Yaskawa INFORM job: LONGPIPE_1.JBI

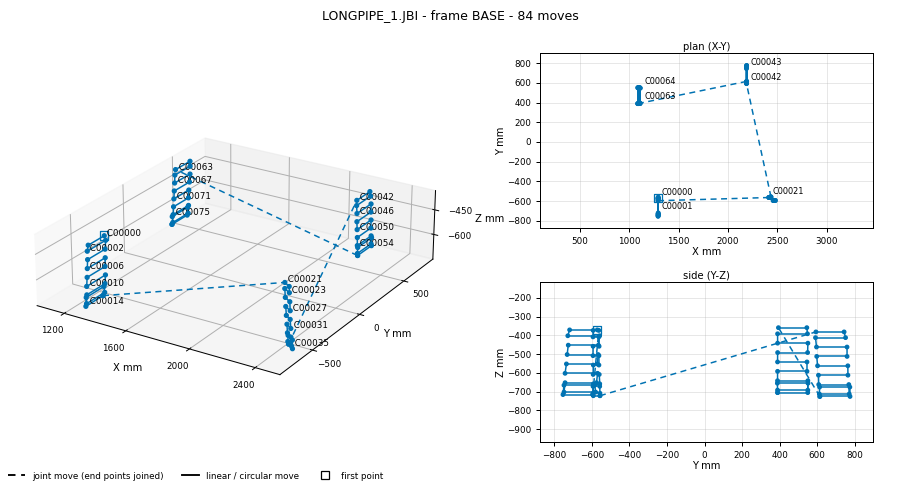
[picture p0: tool path of LONGPIPE_1.JBI in frame BASE, 84 of 89 moves have a stored position in this frame; points joined in program order, loops and branches not executed]
/JOB
//NAME LONGPIPE_1
//POS
///NPOS 84,0,84,0,0,0
///TOOL 1
///POSTYPE BASE
///RECTAN
///RCONF 1,0,0,0,0,0,0,0,0,0,0,0,0,0,0,0,0,0,0,0,0,0,0,0
C00000=1293.713569,-571.374698,-371.239941,175.000000,-89.999999,5.000000
C00001=1293.713569,-718.549324,-371.239941,175.000000,-89.999999,5.000000
C00002=1293.518411,-728.243914,-402.544866,175.000000,-89.999999,5.000000
C00003=1293.518411,-558.764125,-402.544866,175.000000,-89.999999,5.000000
C00004=1292.393979,-565.555949,-452.544866,175.000000,-89.999999,5.000000
C00005=1292.393979,-725.875043,-452.544866,175.000000,-89.999999,5.000000
C00006=1292.721121,-731.714794,-502.544866,175.000000,-89.999999,5.000000
C00007=1292.721121,-566.567624,-502.544866,175.000000,-89.999999,5.000000
C00008=1292.721835,-570.937787,-552.544866,175.000000,-89.999999,5.000000
C00009=1292.721835,-735.641722,-552.544866,175.000000,-89.999999,5.000000
C00010=1293.523260,-742.896244,-602.544866,175.000000,-89.999999,5.000000
C00011=1293.523260,-569.798478,-602.544866,175.000000,-89.999999,5.000000
C00012=1292.629099,-575.385878,-652.544866,175.000000,-89.999999,5.000000
C00013=1292.629099,-742.820182,-652.544866,175.000000,-89.999999,5.000000
C00014=1292.888223,-748.485672,-702.544866,175.000000,-89.999999,5.000000
C00015=1292.888223,-580.024935,-702.544866,175.000000,-89.999999,5.000000
C00016=1292.167541,-584.742252,-665.942326,180.000000,-60.000000,0.000000
C00017=1292.167541,-748.713534,-665.942326,180.000000,-60.000000,0.000000
C00018=1292.184485,-754.080694,-715.942326,180.000000,-60.000000,0.000000
C00019=1292.184485,-595.509845,-715.942326,180.000000,-60.000000,0.000000
C00020=1292.184485,-595.509845,-715.942326,180.000000,-60.000000,0.000000
C00021=2414.469520,-563.186486,-374.006218,175.000000,-89.999999,5.000000
C00022=2458.279331,-593.219364,-374.006218,175.000000,-89.999999,5.000000
C00023=2460.183802,-594.022251,-408.589833,175.000000,-89.999999,5.000000
C00024=2414.262741,-562.730484,-408.589833,175.000000,-89.999999,5.000000
C00025=2417.092851,-561.533351,-458.589833,175.000000,-89.999999,5.000000
C00026=2462.984030,-593.556279,-458.589833,175.000000,-89.999999,5.000000
C00027=2466.185165,-593.992500,-508.589833,175.000000,-89.999999,5.000000
C00028=2420.839516,-562.432648,-508.589833,175.000000,-89.999999,5.000000
C00029=2424.831559,-562.532999,-558.589833,175.000000,-89.999999,5.000000
C00030=2465.448385,-592.380293,-558.589833,175.000000,-89.999999,5.000000
C00031=2470.324386,-593.182778,-608.589833,175.000000,-89.999999,5.000000
C00032=2428.040925,-560.830654,-608.589833,175.000000,-89.999999,5.000000
C00033=2429.847602,-558.174252,-658.589833,175.000000,-89.999999,5.000000
C00034=2470.561816,-591.761141,-658.589833,175.000000,-89.999999,5.000000
C00035=2476.012499,-593.196447,-708.589833,175.000000,-89.999999,5.000000
C00036=2432.039698,-557.009442,-708.589833,175.000000,-89.999999,5.000000
C00037=2434.059154,-558.282965,-671.987293,180.000000,-60.000000,0.000000
C00038=2480.714401,-593.879927,-671.987293,180.000000,-60.000000,0.000000
C00039=2481.009891,-592.462310,-721.987293,180.000000,-60.000000,0.000000
C00040=2436.889101,-556.997461,-721.987293,180.000000,-60.000000,0.000000
C00041=2436.889101,-556.997461,-721.987293,180.000000,-60.000000,0.000000
C00042=2188.305365,593.418636,-381.989438,175.000000,-89.999999,5.000000
C00043=2188.305365,743.516543,-381.989438,175.000000,-89.999999,5.000000
C00044=2189.106018,751.193217,-412.529730,175.000000,-89.999999,5.000000
C00045=2189.106018,591.212146,-412.529730,175.000000,-89.999999,5.000000
C00046=2189.387956,596.556561,-462.529730,175.000000,-89.999999,5.000000
C00047=2189.387956,759.076184,-462.529730,175.000000,-89.999999,5.000000
C00048=2189.662565,759.302992,-512.529730,175.000000,-89.999999,5.000000
C00049=2189.662565,597.699682,-512.529730,175.000000,-89.999999,5.000000
C00050=2189.777671,602.273583,-562.529730,175.000000,-89.999999,5.000000
C00051=2189.777671,763.438563,-562.529730,175.000000,-89.999999,5.000000
C00052=2189.563394,763.900612,-612.529730,175.000000,-89.999999,5.000000
C00053=2189.563394,607.018949,-612.529730,175.000000,-89.999999,5.000000
C00054=2190.031313,608.329641,-662.529730,175.000000,-89.999999,5.000000
C00055=2190.031313,768.620191,-662.529730,175.000000,-89.999999,5.000000
C00056=2189.875845,770.741334,-712.529730,175.000000,-89.999999,5.000000
C00057=2189.875845,611.615028,-712.529730,175.000000,-89.999999,5.000000
C00058=2190.222482,613.157313,-675.927189,180.000000,-60.000000,0.000000
C00059=2190.222482,774.179129,-675.927189,180.000000,-60.000000,0.000000
C00060=2190.098794,775.124391,-725.927189,180.000000,-60.000000,0.000000
C00061=2190.098794,614.285107,-725.927189,180.000000,-60.000000,0.000000
C00062=2190.098794,614.285107,-725.927189,180.000000,-60.000000,0.000000
C00063=1111.787222,393.756921,-359.416126,175.000000,-89.999999,5.000000
C00064=1111.787222,544.977010,-359.416126,175.000000,-89.999999,5.000000
C00065=1110.005604,548.344512,-391.998804,175.000000,-89.999999,5.000000
C00066=1110.005604,389.222439,-391.998804,175.000000,-89.999999,5.000000
C00067=1107.266120,389.333605,-441.998804,175.000000,-89.999999,5.000000
C00068=1107.266120,550.637183,-441.998804,175.000000,-89.999999,5.000000
C00069=1104.078509,549.101244,-491.998804,175.000000,-89.999999,5.000000
C00070=1104.078509,389.470702,-491.998804,175.000000,-89.999999,5.000000
C00071=1101.004161,389.002238,-541.998804,175.000000,-89.999999,5.000000
C00072=1101.004161,545.842938,-541.998804,175.000000,-89.999999,5.000000
C00073=1097.867461,545.873976,-591.998804,175.000000,-89.999999,5.000000
C00074=1097.867461,389.126551,-591.998804,175.000000,-89.999999,5.000000
C00075=1094.734199,388.884036,-641.998804,175.000000,-89.999999,5.000000
C00076=1094.734199,550.514880,-641.998804,175.000000,-89.999999,5.000000
C00077=1091.750483,550.301072,-691.998804,175.000000,-89.999999,5.000000
C00078=1091.750483,388.988649,-691.998804,175.000000,-89.999999,5.000000
C00079=1088.482341,388.038452,-655.396264,180.000000,-60.000000,0.000000
C00080=1088.482341,551.136766,-655.396264,180.000000,-60.000000,0.000000
C00081=1085.230604,549.813872,-705.396264,180.000000,-60.000000,0.000000
C00082=1085.230604,389.311331,-705.396264,180.000000,-60.000000,0.000000
C00083=1085.230604,389.311331,-705.396264,180.000000,-60.000000,0.000000
///TOOL 0
####TOOL####
//INST
///DATE 2022/07/25 12:21
///DATE 2023/06/07 15:00
///ATTR SC,RW
///GROUP1 RB1
///GROUP2 ST1
NOP
MOVJ P009 VJ=15.00
MOVJ C00000 EC00000 VJ=15.0
CALL JOB:SPYON
MOVL C00001 EC00001 V=150.0
MOVL C00002 EC00002 V=150.0
MOVL C00003 EC00003 V=150.0
MOVL C00004 EC00004 V=150.0
MOVL C00005 EC00005 V=150.0
MOVL C00006 EC00006 V=150.0
MOVL C00007 EC00007 V=150.0
MOVL C00008 EC00008 V=150.0
MOVL C00009 EC00009 V=150.0
MOVL C00010 EC00010 V=150.0
MOVL C00011 EC00011 V=150.0
MOVL C00012 EC00012 V=150.0
MOVL C00013 EC00013 V=150.0
MOVL C00014 EC00014 V=150.0
MOVL C00015 EC00015 V=150.0
MOVL C00016 EC00016 V=150.0
MOVL C00017 EC00017 V=150.0
MOVL C00018 EC00018 V=150.0
MOVL C00019 EC00019 V=150.0
CALL JOB:SPYOF
MOVJ P009 VJ=15.00
MOVL C00020 EC00020 V=150.0
MOVJ C00021 EC00021 VJ=15.0
CALL JOB:SPYON
MOVL C00022 EC00022 V=150.0
MOVL C00023 EC00023 V=150.0
MOVL C00024 EC00024 V=150.0
MOVL C00025 EC00025 V=150.0
MOVL C00026 EC00026 V=150.0
MOVL C00027 EC00027 V=150.0
MOVL C00028 EC00028 V=150.0
MOVL C00029 EC00029 V=150.0
MOVL C00030 EC00030 V=150.0
MOVL C00031 EC00031 V=150.0
MOVL C00032 EC00032 V=150.0
MOVL C00033 EC00033 V=150.0
MOVL C00034 EC00034 V=150.0
MOVL C00035 EC00035 V=150.0
MOVL C00036 EC00036 V=150.0
MOVL C00037 EC00037 V=150.0
MOVL C00038 EC00038 V=150.0
MOVL C00039 EC00039 V=150.0
MOVL C00040 EC00040 V=150.0
CALL JOB:SPYOF
MOVJ P009 VJ=15.00
MOVL C00041 EC00041 V=150.0
MOVJ C00042 EC00042 VJ=15.0
CALL JOB:SPYON
MOVL C00043 EC00043 V=150.0
MOVL C00044 EC00044 V=150.0
MOVL C00045 EC00045 V=150.0
MOVL C00046 EC00046 V=150.0
MOVL C00047 EC00047 V=150.0
MOVL C00048 EC00048 V=150.0
MOVL C00049 EC00049 V=150.0
MOVL C00050 EC00050 V=150.0
MOVL C00051 EC00051 V=150.0
MOVL C00052 EC00052 V=150.0
MOVL C00053 EC00053 V=150.0
MOVL C00054 EC00054 V=150.0
MOVL C00055 EC00055 V=150.0
MOVL C00056 EC00056 V=150.0
MOVL C00057 EC00057 V=150.0
MOVL C00058 EC00058 V=150.0
MOVL C00059 EC00059 V=150.0
MOVL C00060 EC00060 V=150.0
MOVL C00061 EC00061 V=150.0
CALL JOB:SPYOF
MOVJ P009 VJ=15.00
MOVL C00062 EC00062 V=150.0
MOVJ C00063 EC00063 VJ=15.0
CALL JOB:SPYON
MOVL C00064 EC00064 V=150.0
MOVL C00065 EC00065 V=150.0
MOVL C00066 EC00066 V=150.0
MOVL C00067 EC00067 V=150.0
MOVL C00068 EC00068 V=150.0
MOVL C00069 EC00069 V=150.0
MOVL C00070 EC00070 V=150.0
MOVL C00071 EC00071 V=150.0
MOVL C00072 EC00072 V=150.0
MOVL C00073 EC00073 V=150.0
MOVL C00074 EC00074 V=150.0
MOVL C00075 EC00075 V=150.0
MOVL C00076 EC00076 V=150.0
MOVL C00077 EC00077 V=150.0
MOVL C00078 EC00078 V=150.0
MOVL C00079 EC00079 V=150.0
MOVL C00080 EC00080 V=150.0
MOVL C00081 EC00081 V=150.0
MOVL C00082 EC00082 V=150.0
CALL JOB:SPYOF
MOVJ P009 VJ=15.00
MOVL C00083 EC00083 V=150.0
END
